// TIA Portal V20 export
TYPE "LConSMC_typeDiamConfig"
// Konfigurationsstruktur des Durchmesserrecheners / Configuration structure of diameter calculation
// stored: Access Published
   STRUCT
      minLineVelocity : LReal := 0.0;   // [m/min oder ft/min] Minimale Bahngeschwindigkeit dass der Durchmesserrechner aktiviert wird / [m/min or ft/min] Minimum web speed to activate the diametet calculation
      minShaftSpeed : LReal := 0.0;   // [min-1] Minimale Drehzahl der Wickelwelle dass der Durchmesserrechner aktiviet wird / [min-1] Minimum winder shaft speed to activate diameter calculation
      minDia : LReal := 0.0;   // [m oder inch] Minimaler Durchmesserwert / [m or inch] Minimum diameter value
      maxDia : LReal := 0.0;   // [m oder inch] Maximaler Durchmesserwert / [m or inch] Maximum diameter value
      webThickness : LReal := 0.0;   // [m oder inch] Materialdicke WIrd für die Berechnungsarten 1&4 benötigt / [m or inch] Web thickness Necessary for the calculation modes 1&4
      useLineAxisActualValues : Bool := TRUE;   // TRUE: Verwende die Istwerte der Bahn zur Durchmesserberechnung. Eingang "lineAxisActualValues" am Wickler FALSE: Verwende die Sollwerte am Eingang "lineAxisMotionVector" / TRUE: Use line actual values (s,v) for the diameter calculation from winder input "lineAxisActualValues" FALSE: Use values from the winder input "lineAxisMotionVector"
      diameterSetValue : LReal := 0.0;   // [m oder inch] Setzwert für den Durchmesser wenn Eingang "setDiameter" am Wicklereingang = TRUE / [m or inch] Diameter set value (If winder input "setDiameter" = TRUE)
      lineFilterTime : Real := 0.0;   // [ms] PT1 Filterzeit für Bahngeschwindigkeit / [ms] PT1 filter time for line velocity
      shaftFilterTime : Real := 0.0;   // [ms] PT1 Filterzeit für Wicklerdrehzahl / [ms] PT1 filter time for winder speed
      measuringRevolutionCount : Real := 4.0;   // Anzahl an Umdrehungen die für die Mittelung des Durchmessers verwenet werden Nur relevant in den Modi Integral (2) und Position (5) / Number of shaft revolutions used for averaging the diameter Only relevant for calculation modes integral (2) and position (5)
      firstDiameterOutput : Real := 0.5;   // Anzahl an Umdrehungen nachdem der erste berechnete Durchmesserwert ausgegeben wird Nur relevant in den Modi Integral (2) und Position (5) / Number of shaft revolutions after which the first diameter value is calculated Only relevant for calculation modes integral (2) and position (5)
      diameterOutputRate : Real := 1.0;   // Anzahl an Umdrehungen nach dem ersten Durchmesserwert nachdem neue berechnete Durchmesserwerte ausgegeben werden Nur relevant in den Modi Integral (2) und Position (5) / Number of shaft revolutions after the first diameter after which a new diameter value is calculated Only relevant for calculation modes integral (2) and position (5)
      lineModLength : Real := 0.0;   // Modulolänge der Bahnachse. 0 = Keine Moduloachse Nur relevant im Mode Position (5) / Modulo length of the line axis. 0 = No modulo axis Only relevant for calculation mode position (5)
      shaftModLength : Real := 0.0;   // Modulolänge der Wicklerachse. 0 = Keine Moduloachse Nur relevant im Mode Position (5) / Modulo length of the winder axis. 0 = No modulo axis Only relevant for calculation mode position (5)
      diameterFilterTime : Real := 0.0;   // [ms] PT1 Filterzeit für Durchmesserausgang / [ms] PT1 filter time for diameter output value
   END_STRUCT;
END_TYPE
